TYPE ST_Floor :
STRUCT
	High,
	Mid,
	Low:BOOL;
END_STRUCT
END_TYPE

(* stored: Version 1.1.0.1, ProductVersion 3.1.4024.11
   DUT ST_Floor: Id {ea72b93e-5f8d-42ad-af7d-054c061a4659} *)
